// TIA Portal V15.1 export
// export: Created 2024-06-21T08:41:08.870147Z, ExportSetting WithDefaults, DisplayName Totally Integrated Automation Portal, DisplayVersion V15.1 Update 5, DisplayName TIA Portal Openness, DisplayVersion V15.1 Update 5, DisplayName SINAMICS Startdrive Advanced, DisplayVersion V15.1, DisplayName G130, G150, S120, S150, SINAMICS MV, S210, DisplayVersion V15.1, DisplayName G110M, G120, G120C, G120D, G120P, DisplayVersion V15.1, DisplayName STEP 7 Professional, DisplayVersion V15.1 Update 5, DisplayName STEP 7 Safety, DisplayVersion V15.1, DisplayName WinCC Professional, DisplayVersion V15.1 Update 5, DisplayName SIMATIC Visualization Architect, DisplayVersion V15.1
FUNCTION "LGBHandHeldHBA-Config" : Void   // FC6712, FBD
TITLE = LGBHandHeldHBA-Config
{ S7_Optimized_Access := 'TRUE' }
AUTHOR : VCG
VERSION : 0.1
// stored: AutoNumber false, IsIECCheckEnabled false, SetENOAutomatically False, UDAEnableTagReadback false
   VAR_INPUT
      C_Device1HighSpeedUsed : Bool;   // Device 1 high speed used
      C_Device2HighSpeedUsed : Bool;   // Device 2 high speed used
      C_Device3HighSpeedUsed : Bool;   // Device 3 high speed used
      C_Device4HighSpeedUsed : Bool;   // Device 4 high speed used
      C_Device5HighSpeedUsed : Bool;   // Device 5 high speed used
      C_Device6HighSpeedUsed : Bool;   // Device 6 high speed used
      C_Device7HighSpeedUsed : Bool;   // Device 7 high speed used
      C_Device8HighSpeedUsed : Bool;   // Device 8 high speed used
      C_Device9HighSpeedUsed : Bool;   // Device 9 high speed used
      C_SpeedValue : Int;   // Speed value for start
      C_MinSpeedValue : Int;   // Minimum speed value
      C_MaxSpeedValue : Int;   // Maximum speed value
      C_SpeedStep : Int;   // Speed step for + or -
   END_VAR
   VAR_IN_OUT
      IO_Config : "HandHeldHBA-Config";   // Config
   END_VAR
BEGIN

REGION Network 1: **** 1 - Inputs **** Move Config
   // Move Config
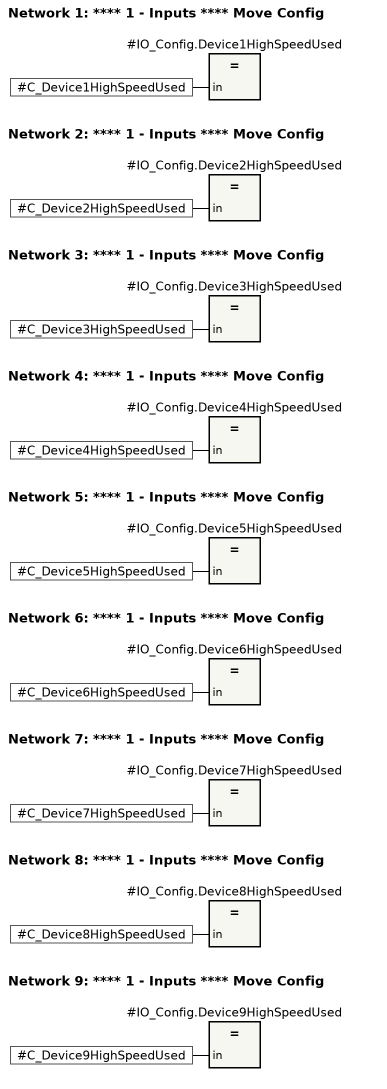
   #IO_Config.Device1HighSpeedUsed := #C_Device1HighSpeedUsed;
END_REGION

REGION Network 2: **** 1 - Inputs **** Move Config
   // Move Config
   #IO_Config.Device2HighSpeedUsed := #C_Device2HighSpeedUsed;
END_REGION

REGION Network 3: **** 1 - Inputs **** Move Config
   // Move Config
   #IO_Config.Device3HighSpeedUsed := #C_Device3HighSpeedUsed;
END_REGION

REGION Network 4: **** 1 - Inputs **** Move Config
   // Move Config
   #IO_Config.Device4HighSpeedUsed := #C_Device4HighSpeedUsed;
END_REGION

REGION Network 5: **** 1 - Inputs **** Move Config
   // Move Config
   #IO_Config.Device5HighSpeedUsed := #C_Device5HighSpeedUsed;
END_REGION

REGION Network 6: **** 1 - Inputs **** Move Config
   // Move Config
   #IO_Config.Device6HighSpeedUsed := #C_Device6HighSpeedUsed;
END_REGION

REGION Network 7: **** 1 - Inputs **** Move Config
   // Move Config
   #IO_Config.Device7HighSpeedUsed := #C_Device7HighSpeedUsed;
END_REGION

REGION Network 8: **** 1 - Inputs **** Move Config
   // Move Config
   #IO_Config.Device8HighSpeedUsed := #C_Device8HighSpeedUsed;
END_REGION

REGION Network 9: **** 1 - Inputs **** Move Config
   // Move Config
   #IO_Config.Device9HighSpeedUsed := #C_Device9HighSpeedUsed;
END_REGION

NETWORK
TITLE = **** 1 Inputs **** Move Config UDT
// Move Config
      L     #C_SpeedValue;
      T     #IO_Config.SpeedValue;
      L     #C_MinSpeedValue;
      T     #IO_Config.MinSpeedValue;
      L     #C_MaxSpeedValue;
      T     #IO_Config.MaxSpeedValue;
      L     #C_SpeedStep;
      T     #IO_Config.SpeedStep;
END_FUNCTION
